% RSLogix 500 project PLC Level 2 Project 4b.RSS, saved by version 8.30.00.16 %
PROJECT "UNTITLED"    % processor: Bul.1763 MicroLogix 1100 Series B %

PROGRAM FILES
  LAD 2 "MAIN"  4 rungs
  LAD 3 "IO CONFIG"  7 rungs
  LAD 4 "CTRL LOGIC"  12 rungs
  LAD 5 "CYCLES"  6 rungs

DATA FILES
  O0 OUTPUT  4 elements
  I1 INPUT  6 elements
  S2 STATUS  66 elements
  B3 BINARY  2 elements
  T4 TIMER  3 elements
  C5 COUNTER  1 elements
  R6 CONTROL  1 elements
  N7 INTEGER  2 elements
  F8 FLOAT  1 elements

LADDER 2 "MAIN"
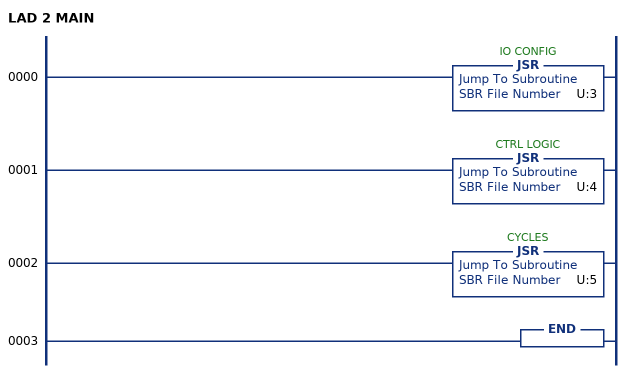
% Rung: 0 %
SOR JSR U:3 EOR
%   U:3  "IO CONFIG" %
% Rung: 1 %
SOR JSR U:4 EOR
%   U:4  "CTRL LOGIC" %
% Rung: 2 %
SOR JSR U:5 EOR
%   U:5  "CYCLES" %
% Rung: 3 %
SOR END EOR

LADDER 3 "IO CONFIG"
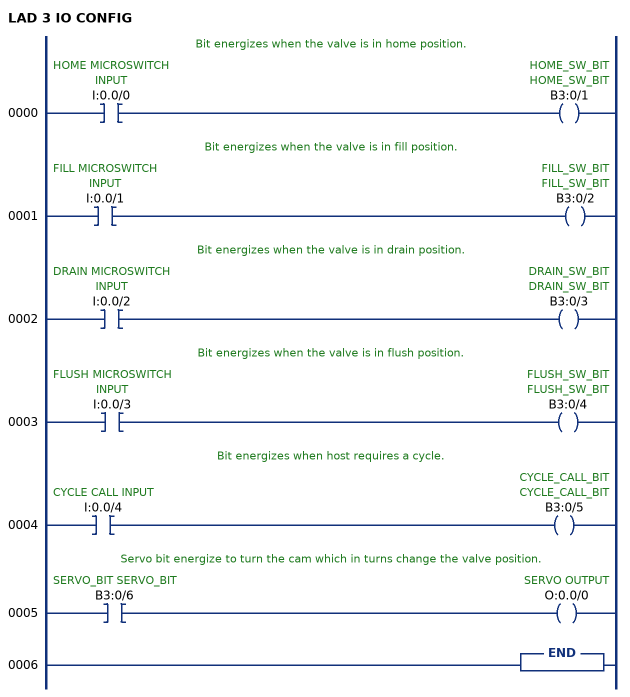
% Rung: 0 %
% Bit energizes when the valve is in home position. %
SOR XIC I:0.0/0 OTE B3:0/1 EOR
%   I:0.0/0  "HOME MICROSWITCH INPUT" %
%   B3:0/1  HOME_SW_BIT  "HOME_SW_BIT" %
% Rung: 1 %
% Bit energizes when the valve is in fill position. %
SOR XIC I:0.0/1 OTE B3:0/2 EOR
%   I:0.0/1  "FILL MICROSWITCH INPUT" %
%   B3:0/2  FILL_SW_BIT  "FILL_SW_BIT" %
% Rung: 2 %
% Bit energizes when the valve is in drain position. %
SOR XIC I:0.0/2 OTE B3:0/3 EOR
%   I:0.0/2  "DRAIN MICROSWITCH INPUT" %
%   B3:0/3  DRAIN_SW_BIT  "DRAIN_SW_BIT" %
% Rung: 3 %
% Bit energizes when the valve is in flush position. %
SOR XIC I:0.0/3 OTE B3:0/4 EOR
%   I:0.0/3  "FLUSH MICROSWITCH INPUT" %
%   B3:0/4  FLUSH_SW_BIT  "FLUSH_SW_BIT" %
% Rung: 4 %
% Bit energizes when host requires a cycle. %
SOR XIC I:0.0/4 OTE B3:0/5 EOR
%   I:0.0/4  "CYCLE CALL INPUT" %
%   B3:0/5  CYCLE_CALL_BIT  "CYCLE_CALL_BIT" %
% Rung: 5 %
% Servo bit energize to turn the cam which in turns change the valve position. %
SOR XIC B3:0/6 OTE O:0.0/0 EOR
%   B3:0/6  SERVO_BIT  "SERVO_BIT" %
%   O:0.0/0  "SERVO OUTPUT" %
% Rung: 6 %
SOR END EOR

LADDER 4 "CTRL LOGIC"
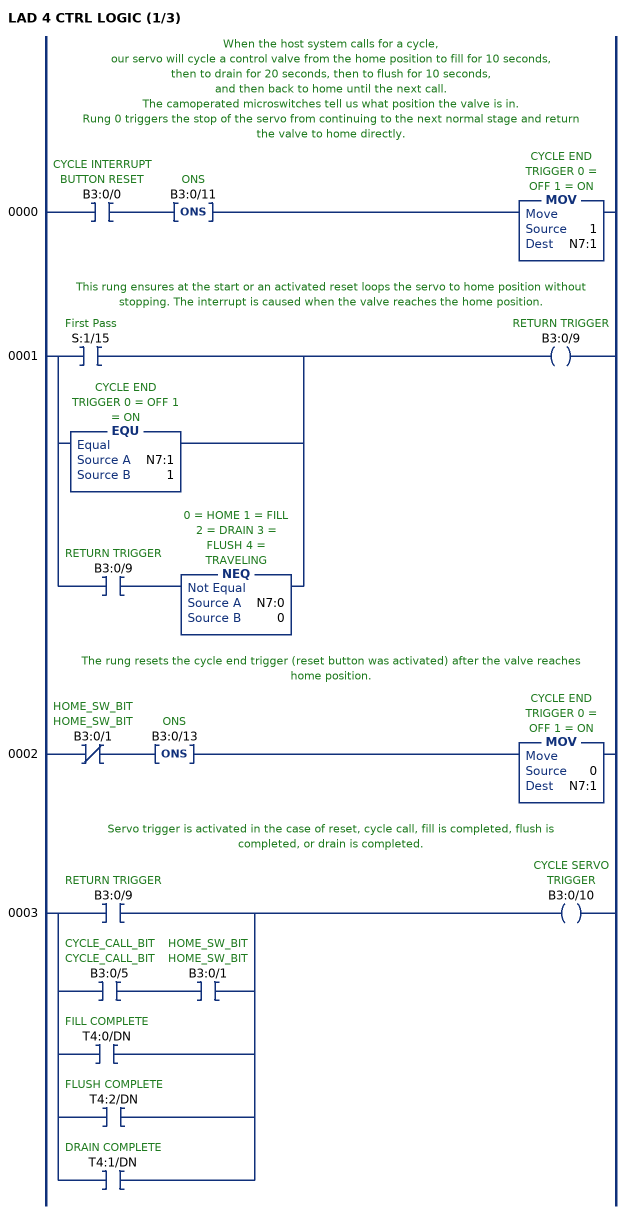
% Rung: 0 %
%  When the host system calls for a cycle, our servo will cycle a control valve from the home position to fill for 10 seconds, then to drain for 20 seconds, then to flush for 10 seconds, and then back to home until the next call.  The camoperated microswitches tell us what position the valve is in. 
% Rung 0 triggers the stop of the servo from continuing to the next normal stage and return the valve to home directly. %
SOR XIC B3:0/0 ONS B3:0/11 MOV 1 N7:1 EOR
%   B3:0/0  RESET  "CYCLE INTERRUPT BUTTON" %
%   B3:0/11  "ONS" %
%   N7:1  "CYCLE END TRIGGER 0 = OFF 1 = ON" %
% Rung: 1 %
% This rung ensures at the start or an activated reset loops the servo to home position without stopping. The interrupt is caused when the valve reaches the home position. %
SOR BST XIC S:1/15 NXB EQU N7:1 1 NXB XIC B3:0/9 NEQ N7:0 0 BND OTE B3:0/9 EOR
%   S:1/15  "First Pass" %
%   N7:1  "CYCLE END TRIGGER 0 = OFF 1 = ON" %
%   B3:0/9  "RETURN TRIGGER" %
%   N7:0  "0 = HOME 1 = FILL 2 = DRAIN 3 = FLUSH 4 = TRAVELING" %
% Rung: 2 %
% The rung resets the cycle end trigger (reset button was activated) after the valve reaches home position. %
SOR XIO B3:0/1 ONS B3:0/13 MOV 0 N7:1 EOR
%   B3:0/1  HOME_SW_BIT  "HOME_SW_BIT" %
%   B3:0/13  "ONS" %
%   N7:1  "CYCLE END TRIGGER 0 = OFF 1 = ON" %
% Rung: 3 %
% Servo trigger is activated in the case of reset, cycle call, fill is completed, flush is completed, or drain is completed. %
SOR BST XIC B3:0/9 NXB XIC B3:0/5 XIC B3:0/1 NXB XIC T4:0/DN NXB XIC T4:2/DN NXB XIC T4:1/DN BND OTE B3:0/10 EOR
%   B3:0/9  "RETURN TRIGGER" %
%   B3:0/5  CYCLE_CALL_BIT  "CYCLE_CALL_BIT" %
%   B3:0/1  HOME_SW_BIT  "HOME_SW_BIT" %
%   T4:0/DN  "FILL COMPLETE" %
%   T4:2/DN  "FLUSH COMPLETE" %
%   T4:1/DN  "DRAIN COMPLETE" %
%   B3:0/10  "CYCLE SERVO TRIGGER" %

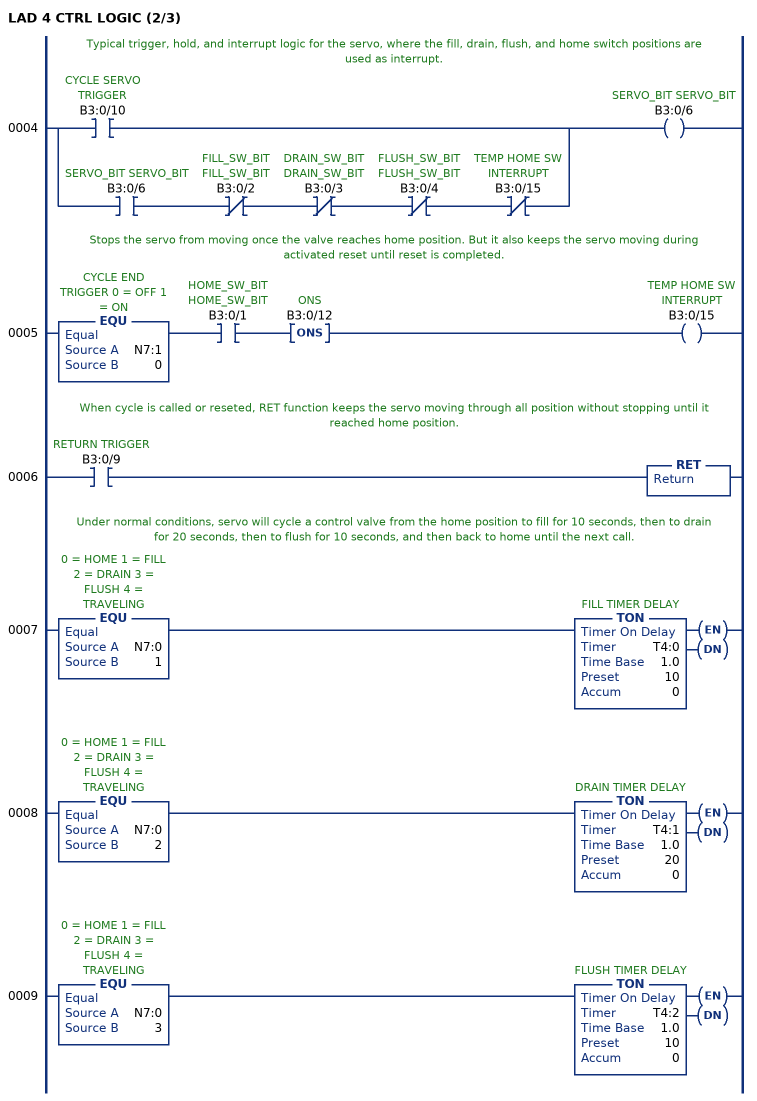
% Rung: 4 %
% Typical trigger, hold, and interrupt logic for the servo, where the fill, drain, flush, and home switch positions are used as interrupt. %
SOR BST XIC B3:0/10 NXB XIC B3:0/6 XIO B3:0/2 XIO B3:0/3 XIO B3:0/4 XIO B3:0/15 BND OTE B3:0/6 EOR
%   B3:0/10  "CYCLE SERVO TRIGGER" %
%   B3:0/6  SERVO_BIT  "SERVO_BIT" %
%   B3:0/2  FILL_SW_BIT  "FILL_SW_BIT" %
%   B3:0/3  DRAIN_SW_BIT  "DRAIN_SW_BIT" %
%   B3:0/4  FLUSH_SW_BIT  "FLUSH_SW_BIT" %
%   B3:0/15  "TEMP HOME SW INTERRUPT" %
% Rung: 5 %
% Stops the servo from moving once the valve reaches home position. But it also keeps the servo moving during activated reset until reset is completed. %
SOR EQU N7:1 0 XIC B3:0/1 ONS B3:0/12 OTE B3:0/15 EOR
%   N7:1  "CYCLE END TRIGGER 0 = OFF 1 = ON" %
%   B3:0/1  HOME_SW_BIT  "HOME_SW_BIT" %
%   B3:0/12  "ONS" %
%   B3:0/15  "TEMP HOME SW INTERRUPT" %
% Rung: 6 %
% When cycle is called or reseted, RET function keeps the servo moving through all position without stopping until it reached home position. %
SOR XIC B3:0/9 RET EOR
%   B3:0/9  "RETURN TRIGGER" %
% Rung: 7 %
% Under normal conditions, servo will cycle a control valve from the home position to fill for 10 seconds, then to drain for 20 seconds, then to flush for 10 seconds, and then back to home until the next call. %
SOR EQU N7:0 1 TON T4:0 1.0 10 0 EOR
%   N7:0  "0 = HOME 1 = FILL 2 = DRAIN 3 = FLUSH 4 = TRAVELING" %
%   T4:0  "FILL TIMER DELAY" %
% Rung: 8 %
SOR EQU N7:0 2 TON T4:1 1.0 20 0 EOR
%   N7:0  "0 = HOME 1 = FILL 2 = DRAIN 3 = FLUSH 4 = TRAVELING" %
%   T4:1  "DRAIN TIMER DELAY" %
% Rung: 9 %
SOR EQU N7:0 3 TON T4:2 1.0 10 0 EOR
%   N7:0  "0 = HOME 1 = FILL 2 = DRAIN 3 = FLUSH 4 = TRAVELING" %
%   T4:2  "FLUSH TIMER DELAY" %

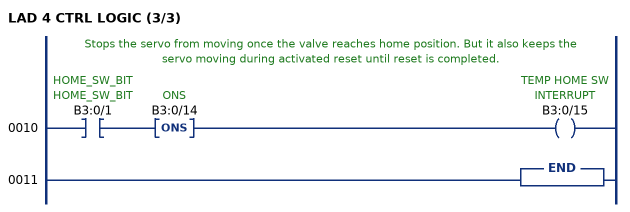
% Rung: 10 %
% Stops the servo from moving once the valve reaches home position. But it also keeps the servo moving during activated reset until reset is completed. %
SOR XIC B3:0/1 ONS B3:0/14 OTE B3:0/15 EOR
%   B3:0/1  HOME_SW_BIT  "HOME_SW_BIT" %
%   B3:0/14  "ONS" %
%   B3:0/15  "TEMP HOME SW INTERRUPT" %
% Rung: 11 %
SOR END EOR

LADDER 5 "CYCLES"
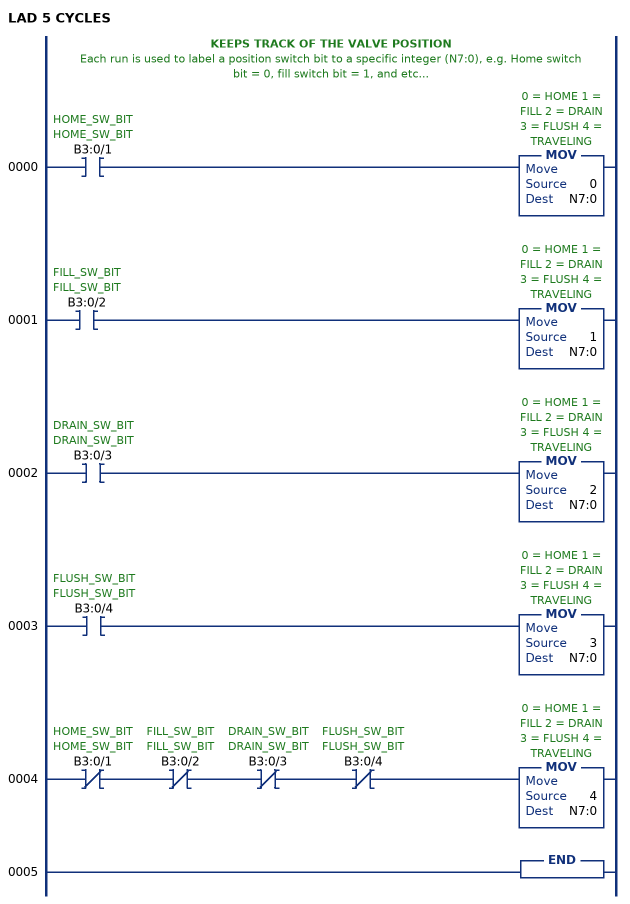
% Rung: 0 %
% TITLE: KEEPS TRACK OF THE VALVE POSITION %
% Each run is used to label a position switch bit to a specific integer (N7:0), e.g. Home switch bit = 0, fill switch bit = 1, and etc... %
SOR XIC B3:0/1 MOV 0 N7:0 EOR
%   B3:0/1  HOME_SW_BIT  "HOME_SW_BIT" %
%   N7:0  "0 = HOME 1 = FILL 2 = DRAIN 3 = FLUSH 4 = TRAVELING" %
% Rung: 1 %
SOR XIC B3:0/2 MOV 1 N7:0 EOR
%   B3:0/2  FILL_SW_BIT  "FILL_SW_BIT" %
%   N7:0  "0 = HOME 1 = FILL 2 = DRAIN 3 = FLUSH 4 = TRAVELING" %
% Rung: 2 %
SOR XIC B3:0/3 MOV 2 N7:0 EOR
%   B3:0/3  DRAIN_SW_BIT  "DRAIN_SW_BIT" %
%   N7:0  "0 = HOME 1 = FILL 2 = DRAIN 3 = FLUSH 4 = TRAVELING" %
% Rung: 3 %
SOR XIC B3:0/4 MOV 3 N7:0 EOR
%   B3:0/4  FLUSH_SW_BIT  "FLUSH_SW_BIT" %
%   N7:0  "0 = HOME 1 = FILL 2 = DRAIN 3 = FLUSH 4 = TRAVELING" %
% Rung: 4 %
SOR XIO B3:0/1 XIO B3:0/2 XIO B3:0/3 XIO B3:0/4 MOV 4 N7:0 EOR
%   B3:0/1  HOME_SW_BIT  "HOME_SW_BIT" %
%   B3:0/2  FILL_SW_BIT  "FILL_SW_BIT" %
%   B3:0/3  DRAIN_SW_BIT  "DRAIN_SW_BIT" %
%   B3:0/4  FLUSH_SW_BIT  "FLUSH_SW_BIT" %
%   N7:0  "0 = HOME 1 = FILL 2 = DRAIN 3 = FLUSH 4 = TRAVELING" %
% Rung: 5 %
SOR END EOR

OTHER DOCUMENTED ADDRESSES
  B3:0/7  "ONS"
  B3:0/8  "ONS"
  B3:1/0  "OFF Cycle Trigger"
  I:0.0/5  "CYCLE RESET INPUT"
  PFILE:6  "Reset Mode"
  U:6  "REST MODE"

DATA TABLE (non-zero values as saved)
DATA T4
% .PRE .ACC %
% T4:0 % 10 0
% T4:1 % 20 0
% T4:2 % 10 0
